TYPE ST_FrameCmd :
STRUCT
	sys   : BYTE;
    sub_s : BYTE;
    dev   : BYTE;
    cmd   : BYTE;
    set   : REAL;
END_STRUCT
END_TYPE

(* stored: Version 1.1.0.1, ProductVersion 3.1.4024.16
   DUT ST_FrameCmd: Id {8aeb47cd-1373-48b6-b28f-415f6889e80d} *)
